{attribute 'qualified_only'}
{attribute 'strict'}
TYPE MoveTypeServo :
(
	None,
	Continuous,
	LinearAbs,
	LinearRel,
	RotaryAbs,
	RotaryRel
);
END_TYPE

(* stored: Version 1.1.0.1, ProductVersion 3.1.4022.11
   DUT MoveTypeServo: Id {3db3393c-2ab8-49c9-8ea3-77907a3ef2b3} *)
